% RSLogix 500 project Project2.RSS, saved by version 8.30.00.16 %
PROJECT "UNTITLED"    % processor: Bul.1763 MicroLogix 1100 Series B %

PROGRAM FILES
  LAD 2 "MAIN"  4 rungs
  LAD 3 "IO"  8 rungs
  LAD 4 "STATE"  7 rungs
  LAD 5 "CTRL"  6 rungs

DATA FILES
  O0 OUTPUT  4 elements
  I1 INPUT  6 elements
  S2 STATUS  66 elements
  B3 BINARY  1 elements
  T4 TIMER  1 elements
  C5 COUNTER  1 elements
  R6 CONTROL  1 elements
  N7 INTEGER  1 elements
  F8 FLOAT  1 elements
  B9 ONESHOT  1 elements

LADDER 2 "MAIN"
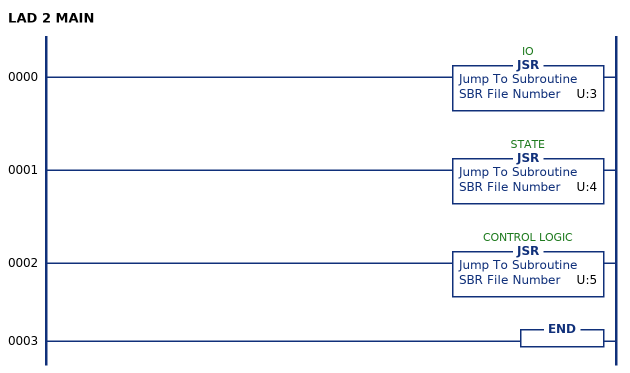
% Rung: 0 %
SOR JSR U:3 EOR
%   U:3  "IO" %
% Rung: 1 %
SOR JSR U:4 EOR
%   U:4  "STATE" %
% Rung: 2 %
SOR JSR U:5 EOR
%   U:5  "CONTROL LOGIC" %
% Rung: 3 %
SOR END EOR

LADDER 3 "IO"
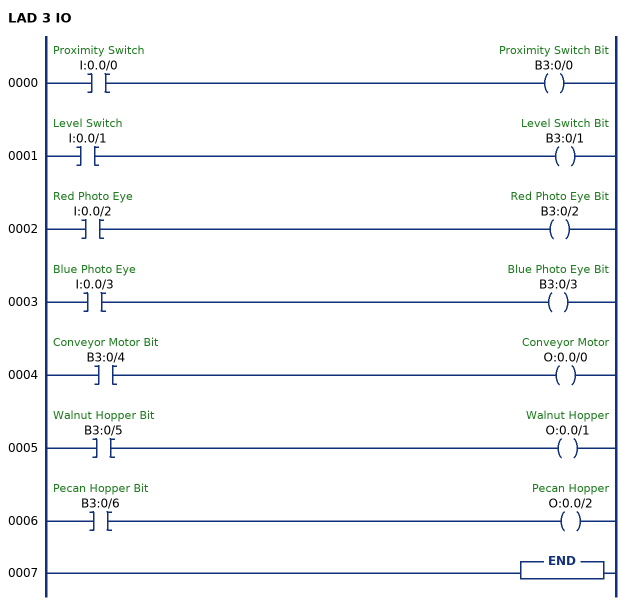
% Rung: 0 %
SOR XIC I:0.0/0 OTE B3:0/0 EOR
%   I:0.0/0  "Proximity Switch" %
%   B3:0/0  "Proximity Switch Bit" %
% Rung: 1 %
SOR XIC I:0.0/1 OTE B3:0/1 EOR
%   I:0.0/1  "Level Switch" %
%   B3:0/1  "Level Switch Bit" %
% Rung: 2 %
SOR XIC I:0.0/2 OTE B3:0/2 EOR
%   I:0.0/2  "Red Photo Eye" %
%   B3:0/2  "Red Photo Eye Bit" %
% Rung: 3 %
SOR XIC I:0.0/3 OTE B3:0/3 EOR
%   I:0.0/3  "Blue Photo Eye" %
%   B3:0/3  "Blue Photo Eye Bit" %
% Rung: 4 %
SOR XIC B3:0/4 OTE O:0.0/0 EOR
%   B3:0/4  "Conveyor Motor Bit" %
%   O:0.0/0  "Conveyor Motor" %
% Rung: 5 %
SOR XIC B3:0/5 OTE O:0.0/1 EOR
%   B3:0/5  "Walnut Hopper Bit" %
%   O:0.0/1  "Walnut Hopper" %
% Rung: 6 %
SOR XIC B3:0/6 OTE O:0.0/2 EOR
%   B3:0/6  "Pecan Hopper Bit" %
%   O:0.0/2  "Pecan Hopper" %
% Rung: 7 %
SOR END EOR

LADDER 4 "STATE"
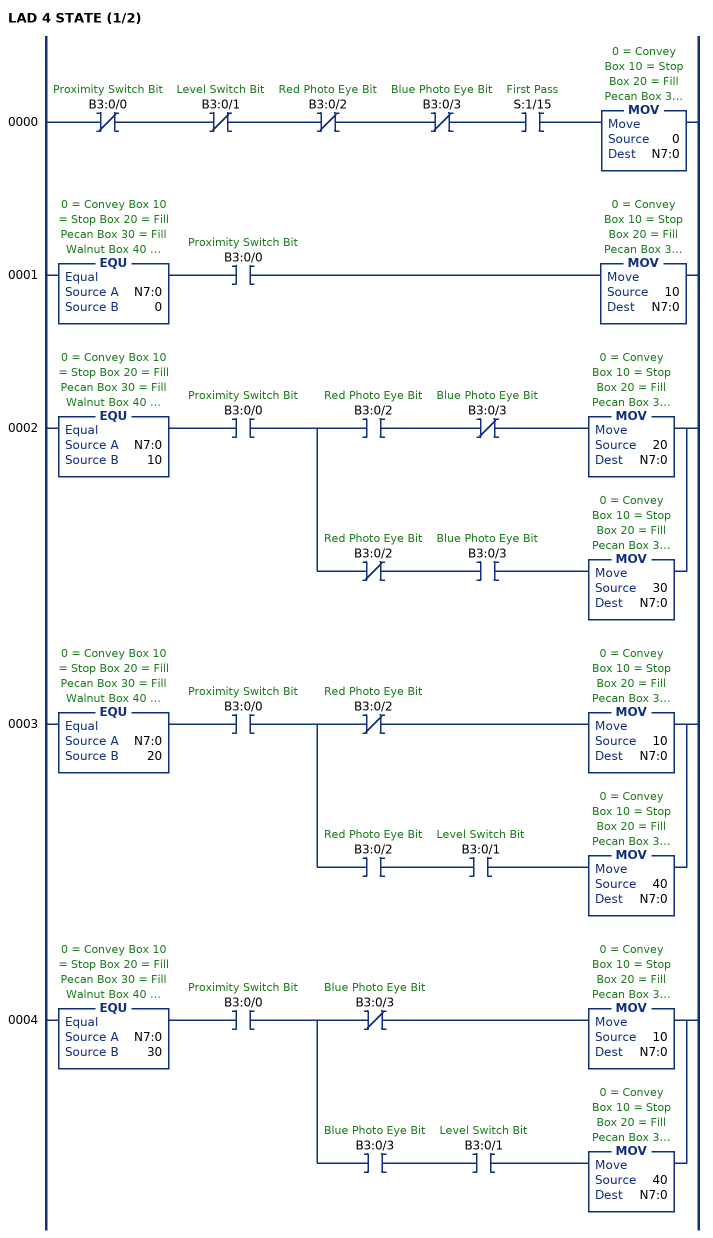
% Rung: 0 %
SOR XIO B3:0/0 XIO B3:0/1 XIO B3:0/2 XIO B3:0/3 XIC S:1/15 MOV 0 N7:0 EOR
%   B3:0/0  "Proximity Switch Bit" %
%   B3:0/1  "Level Switch Bit" %
%   B3:0/2  "Red Photo Eye Bit" %
%   B3:0/3  "Blue Photo Eye Bit" %
%   S:1/15  "First Pass" %
%   N7:0  "0 = Convey Box 10 = Stop Box 20 = Fill Pecan Box 30 = Fill Walnut Box 40 = Unload Box" %
% Rung: 1 %
SOR EQU N7:0 0 XIC B3:0/0 MOV 10 N7:0 EOR
%   N7:0  "0 = Convey Box 10 = Stop Box 20 = Fill Pecan Box 30 = Fill Walnut Box 40 = Unload Box" %
%   B3:0/0  "Proximity Switch Bit" %
% Rung: 2 %
SOR EQU N7:0 10 XIC B3:0/0 BST XIC B3:0/2 XIO B3:0/3 MOV 20 N7:0 NXB XIO B3:0/2 XIC B3:0/3 MOV 30 N7:0 BND EOR
%   N7:0  "0 = Convey Box 10 = Stop Box 20 = Fill Pecan Box 30 = Fill Walnut Box 40 = Unload Box" %
%   B3:0/0  "Proximity Switch Bit" %
%   B3:0/2  "Red Photo Eye Bit" %
%   B3:0/3  "Blue Photo Eye Bit" %
% Rung: 3 %
SOR EQU N7:0 20 XIC B3:0/0 BST XIO B3:0/2 MOV 10 N7:0 NXB XIC B3:0/2 XIC B3:0/1 MOV 40 N7:0 BND EOR
%   N7:0  "0 = Convey Box 10 = Stop Box 20 = Fill Pecan Box 30 = Fill Walnut Box 40 = Unload Box" %
%   B3:0/0  "Proximity Switch Bit" %
%   B3:0/2  "Red Photo Eye Bit" %
%   B3:0/1  "Level Switch Bit" %
% Rung: 4 %
SOR EQU N7:0 30 XIC B3:0/0 BST XIO B3:0/3 MOV 10 N7:0 NXB XIC B3:0/3 XIC B3:0/1 MOV 40 N7:0 BND EOR
%   N7:0  "0 = Convey Box 10 = Stop Box 20 = Fill Pecan Box 30 = Fill Walnut Box 40 = Unload Box" %
%   B3:0/0  "Proximity Switch Bit" %
%   B3:0/3  "Blue Photo Eye Bit" %
%   B3:0/1  "Level Switch Bit" %

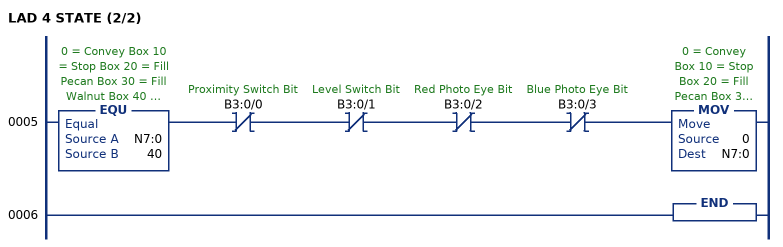
% Rung: 5 %
SOR EQU N7:0 40 XIO B3:0/0 XIO B3:0/1 XIO B3:0/2 XIO B3:0/3 MOV 0 N7:0 EOR
%   N7:0  "0 = Convey Box 10 = Stop Box 20 = Fill Pecan Box 30 = Fill Walnut Box 40 = Unload Box" %
%   B3:0/0  "Proximity Switch Bit" %
%   B3:0/1  "Level Switch Bit" %
%   B3:0/2  "Red Photo Eye Bit" %
%   B3:0/3  "Blue Photo Eye Bit" %
% Rung: 6 %
SOR END EOR

LADDER 5 "CTRL"
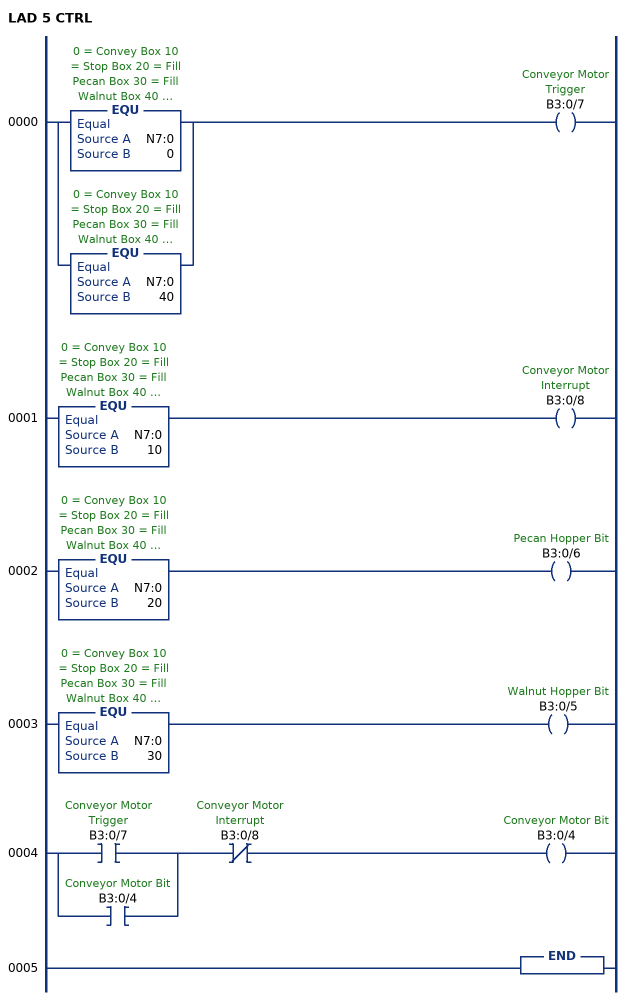
% Rung: 0 %
SOR BST EQU N7:0 0 NXB EQU N7:0 40 BND OTE B3:0/7 EOR
%   N7:0  "0 = Convey Box 10 = Stop Box 20 = Fill Pecan Box 30 = Fill Walnut Box 40 = Unload Box" %
%   B3:0/7  "Conveyor Motor Trigger" %
% Rung: 1 %
SOR EQU N7:0 10 OTE B3:0/8 EOR
%   N7:0  "0 = Convey Box 10 = Stop Box 20 = Fill Pecan Box 30 = Fill Walnut Box 40 = Unload Box" %
%   B3:0/8  "Conveyor Motor Interrupt" %
% Rung: 2 %
SOR EQU N7:0 20 OTE B3:0/6 EOR
%   N7:0  "0 = Convey Box 10 = Stop Box 20 = Fill Pecan Box 30 = Fill Walnut Box 40 = Unload Box" %
%   B3:0/6  "Pecan Hopper Bit" %
% Rung: 3 %
SOR EQU N7:0 30 OTE B3:0/5 EOR
%   N7:0  "0 = Convey Box 10 = Stop Box 20 = Fill Pecan Box 30 = Fill Walnut Box 40 = Unload Box" %
%   B3:0/5  "Walnut Hopper Bit" %
% Rung: 4 %
SOR BST XIC B3:0/7 NXB XIC B3:0/4 BND XIO B3:0/8 OTE B3:0/4 EOR
%   B3:0/7  "Conveyor Motor Trigger" %
%   B3:0/4  "Conveyor Motor Bit" %
%   B3:0/8  "Conveyor Motor Interrupt" %
% Rung: 5 %
SOR END EOR

OTHER DOCUMENTED ADDRESSES
  B9:0/0  "ONS"
